PROGRAM PRG_LIB
VAR
    {attribute 'pytmc' := '
        pv: LIB:
        io: io
    '}
    {attribute 'TcLinkTo' := '.fbLaser.iLaserINT := TIIB[LIB-EL4004-E4]^AO Outputs Channel 1^Analog output;
                              .fbLaser.iShutdownINT := TIIB[LIB-EL4004-E4]^AO Outputs Channel 2^Analog output'}
    fbLIB: FB_REF;
END_VAR

fbLIB.nTransitionAssertionID := 16#6140;
fbLIB.nUnknownAssertionID := 16#6149;

fbLIB.stOut.fPosition := -33.5; // Upper limit
fbLIB.stOut.bUseRawCounts := FALSE;
fbLIB.stOut.nRequestAssertionID := 16#6141;
fbLIB.stOut.stBeamParams := PMPS_GVL.cstFullBeam;
fbLIB.stOut.bValid := TRUE;

fbLIB.stIn.fPosition := -75; // Current position at time of edit
fbLIB.stIn.bUseRawCounts := FALSE;
fbLIB.stIn.nRequestAssertionID := 16#6142;
fbLIB.stIn.stBeamParams := PMPS_GVL.cst0RateBeam;
fbLIB.stIn.bValid := TRUE;

//fbLIB(
//    stYStage := Main.M1,
//    fbArbiter := fbArbiter,
//    fbFFHWO := fbFastFaultOutput1);

END_PROGRAM

(* stored: Version 1.1.0.1, ProductVersion 3.1.4022.18
   POU PRG_LIB: Id {41f87cec-8d4f-488b-ae3e-a2c9e5843eec}, SpecialFunc None *)
